Yaskawa INFORM job: R1_W72(-45,-90)R2.JBI

/JOB
//NAME R1_W72(-45,-90)R2
///FOLDERNAME KRIS-SCIANA
//POS
///NPOS 46,46,0,3,0,0
///TOOL 0
///POSTYPE PULSE
///PULSE
C00000=-100291,-51146,-79231,1033,88265,87213
C00001=-100291,-53738,-49285,1102,68508,87045
C00002=-100261,-52589,-44460,1110,66129,87034
C00003=-99712,-54799,-42787,952,63959,87216
C00004=-99925,-53279,-41211,1022,63773,87136
C00005=-100248,-52046,-42473,1114,65186,87029
C00006=-97451,-51680,-40436,211,64093,88059
C00007=-97263,-52482,-40368,149,63639,88130
C00008=-100239,-51616,-40982,1117,64488,87025
C00009=-100252,-52191,-42992,1113,65430,87029
C00010=-100283,-55028,-57006,1073,72594,87085
C00011=-105536,-81925,-82089,2668,74331,-78427
C00012=-99606,-57790,-58390,866,72020,-76393
C00013=-99356,-58911,-56436,797,70238,-76317
C00014=-99528,-57739,-55221,851,70094,-76380
C00015=-99606,-57531,-56594,872,71047,-76400
C00016=-99710,-56682,-55112,904,70570,-76442
C00017=-99507,-57810,-55028,845,69938,-76374
C00018=-99604,-57511,-56440,872,70964,-76400
C00019=-99614,-57277,-55323,876,70395,-76408
C00020=-99145,-56778,-51373,739,68217,-76254
C00021=-98184,-56617,-50791,435,67936,-75906
C00022=-99614,-56540,-51602,888,68485,-76422
C00023=-99606,-57790,-58390,866,72020,-76393
C00024=-89631,-41013,-57507,2374,78617,-72496
C00025=-89631,-41446,-50339,2416,73987,-72585
C00026=-99891,-48615,-50040,5824,70652,-76293
C00027=-100023,-49746,-50711,5875,70495,-76350
C00028=-100349,-46549,-48840,5964,71008,-76441
C00029=-99774,-50960,-50610,6632,68990,-75291
C00030=-99112,-56968,-51592,9046,64199,-72251
C00031=-99343,-57057,-51554,9138,64153,-72341
C00032=-99465,-56771,-49262,9280,62922,-72490
C00033=-102933,-62363,-48244,10923,59909,-74106
C00034=-99624,-57181,-55073,10007,65604,-71228
C00035=-107649,-61140,-65492,16011,74824,75615
C00036=-107627,-57603,-46892,16933,65566,74318
C00037=-106818,-55773,-41724,16987,63250,74281
C00038=-104140,-55525,-39833,16297,61708,75101
C00039=-106487,-56898,-41551,16985,62526,74298
C00040=-106683,-53850,-39895,16966,63089,74310
C00041=-97681,-55130,-45166,13731,63884,77909
C00042=-99627,-55450,-47389,14246,65390,77352
C00043=-99627,-56586,-52136,14008,67661,77632
C00044=-99623,-55016,-79586,13087,84896,79550
C00045=-92953,-51723,-75150,12718,83736,79808
BC00000=10916,706755,1068222
BC00001=10916,706755,1068222
BC00002=11628,706766,1068222
BC00003=12169,708184,1068222
BC00004=12169,708184,1068222
BC00005=11914,706771,1068222
BC00006=11971,706531,1068222
BC00007=11971,706531,1068222
BC00008=11971,706531,1068222
BC00009=11686,706527,1068222
BC00010=10973,706515,1068222
BC00011=141798,706842,1068222
BC00012=142557,706808,1068222
BC00013=143097,708067,1068222
BC00014=143097,708067,1068222
BC00015=142860,706794,1068222
BC00016=144222,705994,1068222
BC00017=144222,705994,1068222
BC00018=144201,707625,1068222
BC00019=127487,708688,1068222
BC00020=127595,702884,1068222
BC00021=127595,702884,1068222
BC00022=127595,702884,1068222
BC00023=142557,706808,1068222
BC00024=128983,699094,1068222
BC00025=128983,699094,1068222
BC00026=156072,696965,1068222
BC00027=130719,698987,1068222
BC00028=130719,698987,1068222
BC00029=147915,698738,1068222
BC00030=123429,704059,1068222
BC00031=123429,704059,1068222
BC00032=114416,701904,1068222
BC00033=114415,701905,1068218
BC00034=108570,700838,1068222
BC00035=876,712090,1068222
BC00036=876,712085,1068222
BC00037=876,711996,1068222
BC00038=876,711961,1068222
BC00039=876,711961,1068222
BC00040=876,711961,1068222
BC00041=100371,703014,1068222
BC00042=102178,702835,1068222
BC00043=100733,702924,1068222
BC00044=100691,702929,1068222
BC00045=100692,677201,1068222
///POSTYPE BASE
///RECTAN
///RCONF 0,0,0,0,0,0,0,0,0,0,0,0,0,0,0,0,0,0,0,0,0,0,0,0
P00006=0.222,-3.123,-1.508,0.0000,0.0000,0.0000
P00021=-0.225,-6.128,-0.405,0.0000,0.0000,0.0000
P00022=0.222,-3.123,-1.508,0.0000,0.0000,0.0000
//INST
///DATE 2024/07/24 09:23
///ATTR SC,RW
///GROUP1 RB1,BS1
NOP
SFTOF
MOVJ C00000 BC00000 VJ=100.00
MOVJ C00001 BC00001 VJ=100.00
MOVL C00002 BC00002 V=100.0
MOVL C00003 BC00003 V=60.0
REFP 3 C00004 BC00004
CALL JOB:SEARCH-R1
SET P022 P006
SFTON P022
MOVL C00005 BC00005 V=60.0
MOVL C00006 BC00006 V=60.0
REFP 3 C00007 BC00007
CALL JOB:SEARCH-R1
SET P022 P006
SFTON P022
MOVL C00008 BC00008 V=60.0
MOVL C00009 BC00009 V=100.0
MOVJ C00010 BC00010 VJ=100.00
'Path S813
SFTOF
MOVJ C00011 BC00011 VJ=100.00
MOVL C00012 BC00012 V=100.0
MOVL C00013 BC00013 V=60.0
REFP 3 C00014 BC00014
CALL JOB:SEARCH-R1
SET P021 P006
SFTON P021
MOVL C00015 BC00015 V=60.0
MOVL C00016 BC00016 V=60.0
REFP 3 C00017 BC00017
CALL JOB:SEARCH-R1
SET P021 P006
SFTON P021
MOVL C00018 BC00018 V=60.0
MOVL C00019 BC00019 V=100.0
MOVL C00020 BC00020 V=60.0
REFP 3 C00021 BC00021
CALL JOB:SEARCH-R1
SET P021 P006
SFTON P021
MOVL C00022 BC00022 V=60.0
MOVL C00023 BC00023 V=166.7
'Path W108
SFTOF
SFTON P021
MOVJ C00024 BC00024 VJ=100.00
MOVL C00025 BC00025 V=250.0
MACRO1 MJ#(0) ARGF6
MOVL C00026 BC00026 V=100.0 PL=0
REFP 1 C00027 BC00027
REFP 2 C00028 BC00028
ARCON
MOVL C00029 BC00029 V=10.0
MACRO1 MJ#(0) ARGF7
MOVL C00030 BC00030 V=10.8
MOVL C00031 BC00031 V=10.8
MOVL C00032 BC00032 V=10.8
MOVL C00033 BC00033 V=10.8
ARCOF
MOVL C00034 BC00034 V=166.7
SFTOF
'Path W110
SFTOF
SFTON P022
MOVJ C00035 BC00035 VJ=100.00
MOVJ C00036 BC00036 VJ=100.00
MOVL C00037 BC00037 V=250.0
MOVL C00038 BC00038 V=166.7 PL=0
REFP 1 C00039 BC00039
REFP 2 C00040 BC00040
MACRO1 MJ#(0) ARGF9
ARCON
SFTON P021
MOVL C00041 BC00041 V=10.8
ARCOF
MOVL C00042 BC00042 V=166.7
MOVL C00043 BC00043 V=333.3
MOVL C00044 BC00044 V=333.3
SFTOF
MOVJ C00045 BC00045 VJ=100.00
END
